RoboDK station: Motoman-Tests.rdk

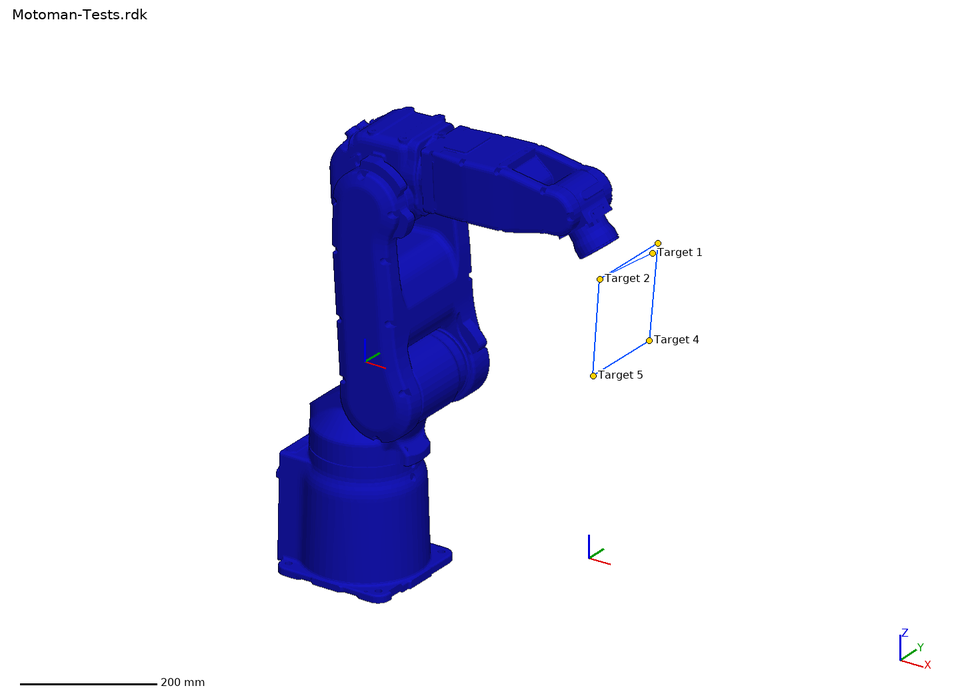
[picture v0: the station drawn from its stored meshes, robots at their saved joint values, targets as dots, program paths as lines]
Station Motoman-Tests. Poses are relative to the parent item; angles as X-Y-Z fixed-axis rotations.
Station parameters (name, value as stored): IO_5, 1
  - frame Motoman MH5F Base at (0, 0, 330) mm
    - robot Motoman MH5F: 6 axes, payload 5 kg, reach 706 mm, repeatability 0.02 mm, weight 27 kg
        modified DH rows (alpha deg, a mm, theta deg, d mm): 0, 0, 0, 330; -90, 88, -90, 0; 0, 310, 0, 0; -90, 40, 0, 305; 90, 0, 0, 0; -90, 0, 0, 80
        base shift (0, 0, -330) mm
        joint limits [-170, -65, -136, -190, -135, -360] to [170, 150, 155, 190, 135, 360]; home [0, 0, 0, 0, 0, 0]; saved at [0, -3.687, -0.703, 0, -56.115, 0]
      - tool Tool, TCP at (-30, 0, 40) mm, rotated rx 0 ry -60 rz 0 deg
    - frame Frame 2 at (399.85, 0, -206.99) mm
      - target Target 1 (joint target) at (113.15, 0, 526.99) mm, rotated rx -180 ry -30 rz 0 deg; joints [0, 0, 0, 0, 0, 0] of Motoman MH5F
      - target Target 2 (Cartesian target) at (18.72, 0, 458.17) mm, rotated rx -180 ry 23.13 rz 0 deg; joints [0, -3.687, -0.703, 0, -56.115, 0] of Motoman MH5F
      - target Target 3 (Cartesian target) at (18.72, 147.32, 458.17) mm, rotated rx -180 ry 23.13 rz 0 deg; joints [21.68, 1.512, 4.395, 15.003, -58.895, -25.526] of Motoman MH5F
      - target Target 4 (Cartesian target) at (3.28, 147.32, 294.99) mm, rotated rx -180 ry 23.13 rz 0 deg; joints [22.53, 1.554, -26.448, 27.261, -30.126, -42.381] of Motoman MH5F
      - target Target 5 (Cartesian target) at (3.28, 4.68, 294.99) mm, rotated rx -180 ry 23.13 rz 0 deg; joints [0.755, -3.909, -31.79, 1.061, -25.256, -1.564] of Motoman MH5F
  - program Program (19 instructions, listed below)
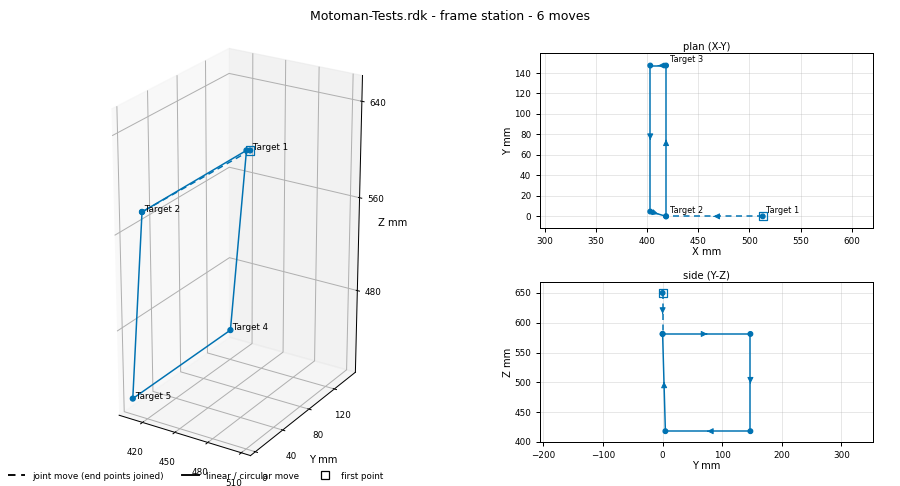
[picture p0: tool path of Motoman-Tests.rdk in frame station, 6 of 6 moves have a stored position in this frame; points joined in program order, loops and branches not executed]

--- program Program (robot Motoman MH5F) ---
  Set Ref.: Frame 2
  Set Tool: Tool 1
  Set speed (100.0 mm/s)
  MoveJ (Target 1)
  MoveJ (Target 2)
  Pause 500 ms
  MoveL (Target 3)
  MoveL (Target 4)
  Print: Stop the robot until the user wants to continue
  Remove next line to prevent ...: Remove next line to prevent the robot from stopping
  Stop
  Print: Running program Prog2
  Call Subprog
  MoveL (Target 5)
  Print: Set Digital Output 5 to ON
  Set IO_5=1
  MoveL (Target 2)
  Print: Wait for digital input 5 to turn ON
  Wait IO_5=1
